INTERFACE I_Color

METHOD M_Fill : BOOL
VAR_INPUT
END_VAR
END_METHOD

END_INTERFACE

(* stored: Version 1.1.0.1, ProductVersion 3.1.4024.12
   Itf I_Color: Id {5c158fde-0479-4e0d-8bed-0812c766e8db}
   Method M_Fill: Id {b5d0011c-4148-42c3-bb9e-200daf9bc97a} *)
